KUKA KRL program: RSI_PathControl_1.src, RSI_PathControl_1.dat

--- RSI_PathControl_1.src ---
&ACCESS RVP
&REL 24
&PARAM EDITMASK = *
&PARAM TEMPLATE = C:\KRC\Roboter\Template\vorgabe
&PARAM DISKPATH = KRC:\R1
DEF RSI_PathControl_1()
   ;FOLD INI;%{PE}
      ;FOLD BASISTECH INI
         GLOBAL INTERRUPT DECL 3 WHEN $STOPMESS==TRUE DO IR_STOPM ( )
         INTERRUPT ON 3
         BAS (#INITMOV,0 )
      ;ENDFOLD (BASISTECH INI)
      ;FOLD USER INI
         ;Make your modifications here
      ;ENDFOLD (USER INI)
   ;ENDFOLD (INI)

   ; Declaration of KRL variables
   ;DECL INT ret        ; Return value for RSI commands
   ;DECL INT container  ; Container ID
   ;DECL INT step       ; Current waypoint step
   ;DECL INT movecorr_flag
   ; Move to home position

   PTP {A1 0, A2 -90, A3 90, A4 0, A5 0, A6 0}

   ; Create RSI Context
   ret = RSI_CREATE("PathControl", container)
   IF (ret <> RSIOK) THEN
      HALT
   ENDIF

   $ANOUT[1]=99
   ; Start RSI execution in RELATIVE mode for smaller corrections
   ret = RSI_ON(#RELATIVE, , ,#BASE)

   IF (ret <> RSIOK) THEN
      HALT
   ENDIF

   LOOP



      IF  ( $ANOUT[1]==1 ) THEN

         step=1
         ret=RSI_SETPUBLICPAR(container,"step","Value", step)
         IF (ret <> RSIOK) THEN
            HALT
         ENDIF
         PTP {A1 30, A2 -90, A3 90, A4 0, A5 90, A6 0}

         ;ENDFOLD
         step=2
         ret=RSI_SETPUBLICPAR(container,"step","Value", step)
         IF (ret <> RSIOK) THEN
            HALT
         ENDIF
         ;FOLD PTP P3 CONT Vel=100 % PDAT1 Tool[1] Base[0] ;%{PE}
            ;FOLD Parameters ;%{h}
               ;Params IlfProvider=kukaroboter.basistech.inlineforms.movement.old; Kuka.IsGlobalPoint=False; Kuka.PointName=P3; Kuka.BlendingEnabled=True; Kuka.MoveDataPtpName=PDAT1; Kuka.VelocityPtp=100; Kuka.CurrentCDSetIndex=0; Kuka.MovementParameterFieldEnabled=True; IlfCommand=PTP
            ;ENDFOLD

            $BWDSTART = FALSE
            PDAT_ACT = PPDAT1
            FDAT_ACT = FP3
            BAS(#PTP_PARAMS, 100.0)
            SET_CD_PARAMS (0)
            PTP XP3 C_Dis

         ;ENDFOLD
         step=3
         ret=RSI_SETPUBLICPAR(container,"step","Value", step)
         IF (ret <> RSIOK) THEN
            HALT
         ENDIF

         ;FOLD LIN P2 CONT Vel=2 m/s CPDAT1 Tool[1] Base[0] ;%{PE}
            ;FOLD Parameters ;%{h}
               ;Params IlfProvider=kukaroboter.basistech.inlineforms.movement.old; Kuka.IsGlobalPoint=False; Kuka.PointName=P2; Kuka.BlendingEnabled=True; Kuka.MoveDataName=CPDAT1; Kuka.VelocityPath=2; Kuka.CurrentCDSetIndex=0; Kuka.MovementParameterFieldEnabled=True; IlfCommand=LIN
            ;ENDFOLD
            $BWDSTART = FALSE
            LDAT_ACT = LCPDAT1
            FDAT_ACT = FP2
            BAS(#CP_PARAMS, 2.0)
            SET_CD_PARAMS (0)
            LIN XP2 C_Dis C_Dis
         ;ENDFOLD

         step=4
         ret=RSI_SETPUBLICPAR(container,"step","Value", step)
         IF (ret <> RSIOK) THEN
            HALT
         ENDIF
         PTP {A1 30, A2 -90, A3 90, A4 0, A5 90, A6 0}

         $ANOUT[1]=99

         ;FOLD WAIT Time= 1.0 sec ;%{PE}
            ;FOLD Parameters ;%{h}
               ;Params IlfProvider=kukaroboter.basistech.inlineforms.logics.wait; Time=1.0
            ;ENDFOLD
            WAIT SEC 1.0
         ;ENDFOLD

      ENDIF

      IF  ( $ANOUT[1]==2 ) THEN

         step=5
         ret=RSI_SETPUBLICPAR(container,"step","Value", step)
         IF (ret <> RSIOK) THEN
            HALT
         ENDIF
         PTP {A1 0, A2 -75, A3 90, A4 -90, A5 90, A6 100}

         step=6
         ret=RSI_SETPUBLICPAR(container,"step","Value", step)
         IF (ret <> RSIOK) THEN
            HALT
         ENDIF

         ;FOLD WAIT Time= 5.0 sec ;%{PE}
            ;FOLD Parameters ;%{h}
               ;Params IlfProvider=kukaroboter.basistech.inlineforms.logics.wait; Time=5.0
            ;ENDFOLD
            WAIT SEC 5.0
         ;ENDFOLD

         movecorr_flag=1
         ret=RSI_SETPUBLICPAR(container,"movecorr_flag","Value", movecorr_flag)
         IF (ret <> RSIOK) THEN
            HALT
         ENDIF
         ; Sensor guided movement
         RSI_MOVECORR()

         movecorr_flag=0
         ret=RSI_SETPUBLICPAR(container,"movecorr_flag","Value", movecorr_flag)
         IF (ret <> RSIOK) THEN
            HALT
         ENDIF

         ;FOLD WAIT Time= 1.0 sec ;%{PE}
            ;FOLD Parameters ;%{h}
               ;Params IlfProvider=kukaroboter.basistech.inlineforms.logics.wait; Time=1.0
            ;ENDFOLD
            WAIT SEC 1.0
         ;ENDFOLD

         movecorr_flag=1
         ret=RSI_SETPUBLICPAR(container,"movecorr_flag","Value", movecorr_flag)
         IF (ret <> RSIOK) THEN
            HALT
         ENDIF
         ; Sensor guided movement
         RSI_MOVECORR()
         movecorr_flag=0
         ret=RSI_SETPUBLICPAR(container,"movecorr_flag","Value", movecorr_flag)
         IF (ret <> RSIOK) THEN
            HALT
         ENDIF

         ;FOLD WAIT Time= 1.0 sec ;%{PE}
            ;FOLD Parameters ;%{h}
               ;Params IlfProvider=kukaroboter.basistech.inlineforms.logics.wait; Time=1.0
            ;ENDFOLD
            WAIT SEC 1.0
         ;ENDFOLD

         $ANOUT[1]=99

         ;FOLD WAIT Time= 1.0 sec ;%{PE}
            ;FOLD Parameters ;%{h}
               ;Params IlfProvider=kukaroboter.basistech.inlineforms.logics.wait; Time=1.0
            ;ENDFOLD
            WAIT SEC 1.0
         ;ENDFOLD

         ENDIF


      IF  ( $ANOUT[1] <> 1) THEN


         IF  ( $ANOUT[1] <> 2 ) THEN
            $ANOUT[1] = 99
            WAIT SEC 1.0
         ENDIF

      ENDIF
   ENDLOOP

   ; Turn off RSI
   ret = RSI_OFF()
   IF (ret <> RSIOK) THEN
      HALT
   ENDIF

   PTP {A1 0, A2 -90, A3 90, A4 0, A5 90, A6 0}

END

--- RSI_PathControl_1.dat ---
&ACCESS  RVP
&PARAM EDITMASK = *
&PARAM TEMPLATE = C:\KRC\Roboter\Template\vorgabe
&PARAM DISKPATH = KRC:\R1
&REL 19
DEFDAT  RSI_PATHCONTROL_1
;FOLD EXTERNAL DECLARATIONS;%{PE}%MKUKATPBASIS,%CEXT,%VCOMMON,%P
;FOLD BASISTECH EXT;%{PE}%MKUKATPBASIS,%CEXT,%VEXT,%P
EXT  BAS (BAS_COMMAND  :IN,REAL  :IN )
DECL INT SUCCESS
;ENDFOLD (BASISTECH EXT)
;FOLD USER EXT;%{E}%MKUKATPUSER,%CEXT,%VEXT,%P
;Make your modifications here
;ENDFOLD (USER EXT)
;ENDFOLD (EXTERNAL DECLARATIONS)

; Variable declarations
DECL INT ret
DECL INT container
DECL INT step
DECL INT movecorr_flag
DECL INT routine_num

DECL E6POS XP1={X 1798.70654,Y 0.000902908039,Z 1837.39172,A -179.999985,B -2.28500152,C -179.999924,S 2,T 35,E1 0.0,E2 0.0,E3 0.0,E4 0.0,E5 0.0,E6 0.0}
DECL E6POS XP2={X 2006.20398,Y 0.00138249062,Z 1522.22,A 179.999771,B -13.7302580,C -179.999817,S 2,T 35,E1 0.0,E2 0.0,E3 0.0,E4 0.0,E5 0.0,E6 0.0}
DECL FDAT FP2={TOOL_NO 1,BASE_NO 0,IPO_FRAME #BASE,POINT2[] " "}
DECL LDAT LCPDAT1={VEL 2.00000,ACC 100.000,APO_DIST 500.000,APO_FAC 50.0000,AXIS_VEL 100.000,AXIS_ACC 100.000,ORI_TYP #VAR,CIRC_TYP #BASE,JERK_FAC 50.0000,GEAR_JERK 100.000,EXAX_IGN 0,CB {AUX_PT {ORI #CONSIDER,E1 #CONSIDER,E2 #CONSIDER,E3 #CONSIDER,E4 #CONSIDER,E5 #CONSIDER,E6 #CONSIDER},TARGET_PT {ORI #INTERPOLATE,E1 #INTERPOLATE,E2 #INTERPOLATE,E3 #INTERPOLATE,E4 #INTERPOLATE,E5 #INTERPOLATE,E6 #INTERPOLATE}}}
DECL MODULEPARAM_T LAST_TP_PARAMS = {PARAMS[] "Kuka.PointName=P3; Kuka.FrameData.base_no=0; Kuka.FrameData.tool_no=1; Kuka.FrameData.ipo_frame=#BASE; Kuka.FrameData.point2=; Kuka.isglobalpoint=False; Kuka.MoveDataName=CPDAT1; Kuka.MovementData.cb={AUX_PT {ORI #CONSIDER,E1 #CONSIDER,E2 #CONSIDER,E3 #CONSIDER,E4 #CONSIDER,E5 #CONSIDER,E6 #CONSIDER},TARGET_PT {ORI #INTERPOLATE,E1 #INTERPOLATE,E2 #INTERPOLATE,E3 #INTERPOLATE,E4 #INTERPOLATE,E5 #INTERPOLATE,E6 #INTERPOLATE}}; Kuka.MovementData.apo_fac=50; Kuka.MovementData.apo_dist=500; Kuka.MovementData.axis_acc=100; Kuka.MovementData.axis_vel=100; Kuka.MovementData.circ_typ=#BASE; Kuka.MovementData.jerk_fac=50; Kuka.MovementData.ori_typ=#VAR; Kuka.MovementData.vel=100; Kuka.MovementData.acc=100; Kuka.MovementData.exax_ign=0; Kuka.VelocityPath=2; Kuka.BlendingEnabled=True; Kuka.APXEnabled=False; Kuka.CurrentCDSetIndex=0; Kuka.MoveDataPtpName=PDAT1; Kuka.MovementDataPdat.apo_mode=#CDIS; Kuka.MovementDataPdat.apo_dist=500; Kuka.VelocityPtp=100; Kuka.Analog.Channel=1; Kuka.Analog.Value=1"}
DECL E6POS XP3={X 1929.01013,Y 0.00523620285,Z 1634.67773,A 179.999741,B -9.58288288,C -179.999786,S 2,T 35,E1 0.0,E2 0.0,E3 0.0,E4 0.0,E5 0.0,E6 0.0}
DECL FDAT FP3={TOOL_NO 1,BASE_NO 0,IPO_FRAME #BASE,POINT2[] " "}
DECL PDAT PPDAT1={VEL 100.000,ACC 100.000,APO_DIST 500.000,APO_MODE #CDIS,GEAR_JERK 100.000,EXAX_IGN 0}
ENDDAT
